(* CoDeSys 2.3 export: PV_REQ.EXP *)

(* Data type *)
TYPE PV_REQ :
	(
	PV_NONE_REQ := 0,
	PV_ISOLATE_REQ,
	PV_PUMP_REQ,
	PV_VENT_REQ
	);
END_TYPE
